{attribute 'qualified_only'}
{attribute 'strict'}
{attribute 'to_string'}
TYPE E_LogLevel :
(
    Verbose 	:= 1,
    Info  		:= 2,
    Warning  	:= 3,
    Error 		:= 4,
    Critical 	:= 5
);
END_TYPE

(* stored: Version 1.1.0.1
   DUT E_LogLevel: Id {f5f9d77b-25ca-489c-8389-9e110ddcd81a} *)
